(* PLC project Unnamed, Unknown Unnamed 1 *)
(* stored: creationDateTime 2021-05-11T15:41:27, modificationDateTime 2021-08-18T14:10:57 *)

PROGRAM CD_LV_PLC
  VAR
    TIME_IN AT %MD0 : REAL;
    TIME_OUT AT %MD1 : REAL;
    CD_Level AT %MD2 : REAL;
    RX_Power AT %MD3 : REAL;
    CE_Pump_Speed_1 AT %MD4 : REAL;
    CE_Pump_Speed_2 AT %MD5 : REAL;
    CE_Pump_Speed_3 AT %MD6 : REAL;
    CE_Pump_OnOff_1 AT %MD7 : REAL := 1.0;
    CE_Pump_OnOff_2 AT %MD8 : REAL := 1.0;
    CE_Pump_OnOff_3 AT %MD9 : REAL := 0.0;
    MANIPIO_CONTROL AT %MD10 : REAL := 0.0;
    KPI AT %MD11 : REAL := -100.0;
    Ti AT %MD12 : REAL := 60.0;
    SET_POINT AT %MD13 : REAL := 1.0;
    INIT AT %MD14 : REAL := 90.0;
  END_VAR
  VAR
    INTEGRAL0 : INTEGRAL;
  END_VAR
  VAR  (* added by the conversion: wires and edge detectors of the diagram *)
    _MUL7_OUT : REAL;
    _LIMIT18_OUT : ANY;
    _ADD14_OUT : ANY;
    _SEL23_OUT : REAL;
  END_VAR

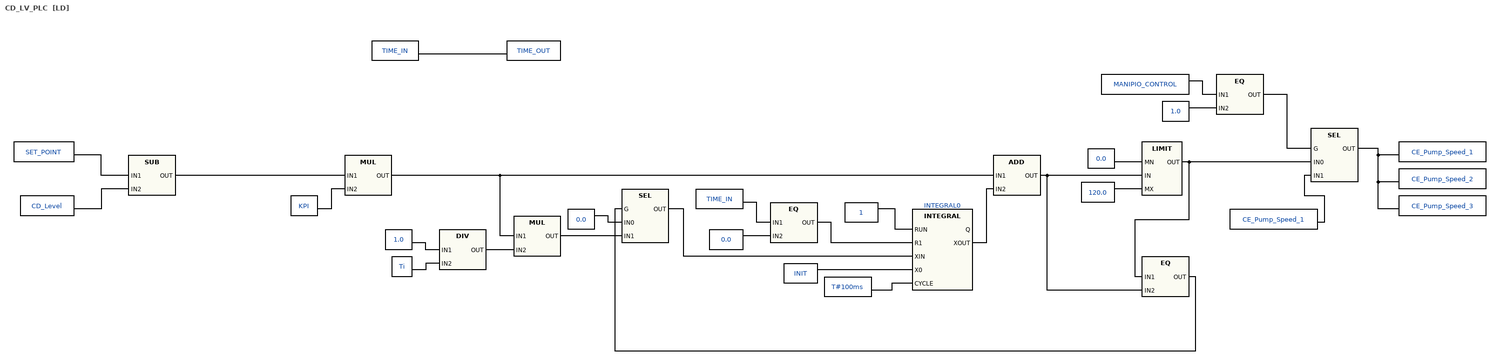
(* LD diagram, written out as Structured Text *)
TIME_OUT := TIME_IN;
_MUL7_OUT := (SET_POINT - CD_Level) * KPI;
INTEGRAL0(RUN := 1, R1 := TIME_IN = 0.0, XIN := SEL(_LIMIT18_OUT = _ADD14_OUT, 0.0, _MUL7_OUT * (1.0 / Ti)), X0 := INIT, CYCLE := T#100ms);
_ADD14_OUT := _MUL7_OUT + INTEGRAL0.XOUT;
_LIMIT18_OUT := LIMIT(0.0, _ADD14_OUT, 120.0);
_SEL23_OUT := SEL(MANIPIO_CONTROL = 1.0, _LIMIT18_OUT, CE_Pump_Speed_1);
CE_Pump_Speed_1 := _SEL23_OUT;
CE_Pump_Speed_2 := _SEL23_OUT;
CE_Pump_Speed_3 := _SEL23_OUT;
END_PROGRAM

CONFIGURATION Config0
  RESOURCE Res0 ON PLC
    TASK task0(INTERVAL := T#100ms, PRIORITY := 0);
    PROGRAM instance0 WITH task0 : CD_LV_PLC;
  END_RESOURCE
END_CONFIGURATION
